// TIA Portal V20 export
FUNCTION "RealBlockName" : Void   // FC17, LAD
BEGIN

REGION Network 1
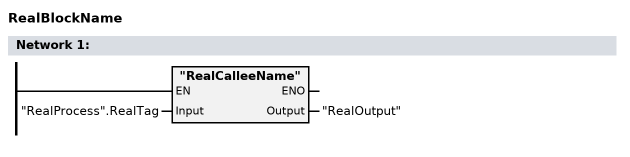
   RUNG wire#powerrail
      "RealCalleeName"(Input := "RealProcess".RealTag, Output => "RealOutput")
   END_RUNG
   // the same network as SCL:
   "RealCalleeName"(Input := "RealProcess".RealTag, Output => "RealOutput");
END_REGION
END_FUNCTION
